FUNCTION F_GetConnectionColor : E_HMI_COLORS
VAR_INPUT
    bConnected : BOOL;
END_VAR
VAR
END_VAR

IF bConnected THEN
    F_GetConnectionColor := E_HMI_COLORS.GREEN;
ELSE
    F_GetConnectionColor := E_HMI_COLORS.RED;
END_IF

END_FUNCTION

(* stored: Version 1.1.0.1, ProductVersion 3.1.4024.14
   POU F_GetConnectionColor: Id {dd8e510c-e6ff-4a9d-9149-cc30bf7be75c}, SpecialFunc None *)
